TYPE ST_LAB_PackData_1 :
STRUCT
	sPackCode				: T_MaxString;
	nPackStatus				: INT;
	nPackRejectID			: UINT;
END_STRUCT
END_TYPE

(* stored: Version 1.1.0.1
   DUT ST_LAB_PackData_1: Id {8cb6e681-cc6f-4273-b632-404c276f2e8d} *)
